TYPE TYP_ALARM_HISTORY_ENTRY :
STRUCT
	Timestamp : DT;
	Name : STRING;
	Message : STRING;
	PreviousState : STRING;
	NewState : STRING;
	Code : DINT;
	Priority : INT;
END_STRUCT
END_TYPE

(* stored: Version 1.1.0.1, ProductVersion 3.1.4024.12
   DUT TYP_ALARM_HISTORY_ENTRY: Id {ffd98be1-0290-4cde-851c-14a233c95d34} *)
